FUNCTION_BLOCK Test_TStreamBufferResizes EXTENDS T_UnitTestBase
VAR
    Stream : T_Stream(StreamLength := 2);
END_VAR

Stream.Init(2);

Stream.Add_INT(1234);
Stream.Add_INT(1235);
Stream.Add_INT(1236);
Stream.Add_INT(1237);

Assertion.AssertEquals_UDINT(Expected     := 8,
                             Actual       := Stream.Position,
                             VariableName := 'Stream.Position');

Assertion.AssertEquals_UDINT(Expected     := 8,
                             Actual       := Stream.StreamLength,
                             VariableName := 'Stream.StreamLength');

Stream.Seek(0);

Assertion.AssertEquals_INT(Expected     := 1234,
                           Actual       := Stream.Read_INT(),
                           VariableName := 'Stream.ReadInt()');

Assertion.AssertEquals_UDINT(Expected     := 2,
                             Actual       := Stream.Position,
                             VariableName := 'Stream.Position');

TestFinished();

END_FUNCTION_BLOCK

(* stored: Version 1.1.0.1, ProductVersion 3.1.4024.6
   POU Test_TStreamBufferResizes: Id {c192b989-d352-4cfc-9e66-f8073ecd67eb}, SpecialFunc None *)
